FUNCTION_BLOCK AxisVelocityTestSuite 
VAR
	StubAxis : AXIS_REF;
	iStubTask : I_Task;
	TestAxisVelo : MoveVeloTask := (AxisRef := StubAxis);
	ObjTestSuite : TestSuite<TestSuiteParameter.MaxTestCount>('C:\ProgramData\Beckhoff\TwinCAT\3.1\Boot\Object_Tests.xml') := (TestSuiteName := 'Object Test Suite');
END_VAR

DoesTaskAcceptAcceleration_Test();
DoesTaskAcceptDeceleration_Test();
DoesTaskAcceptJerk_Test();
DoesTaskRejectAZeroVelocity_Test();
DoesTaskRejectNegativeAccell_Test();
DoesTaskRejectNegativeDecel_Test();
DoesTaskRejectNegativeJerk_Test();
DoesTaskRejectNegativeVelocity_Test();

METHOD DoesTaskAcceptAcceleration_Test
VAR_INST
	Expected : BOOL := TRUE;
	Actual	 : BOOL;
END_VAR
IF ObjTestSuite.Test(__POUNAME()).ExecuteTest() THEN
	TestAxisVelo.Acceleration := 1.0;
	Actual := TestAxisVelo.Acceleration = 1.0;
	ObjTestSuite.Test(__POUNAME()).AssertEqual(Expected, Actual);
	TestAxisVelo.Acceleration := 0.0;
	TestAxisVelo.Abort();
END_IF
END_METHOD

METHOD DoesTaskAcceptDeceleration_Test
VAR_INST
	Expected : BOOL := TRUE;
	Actual	 : BOOL;
END_VAR
IF ObjTestSuite.Test(__POUNAME()).ExecuteTest() THEN
	TestAxisVelo.Deceleration := 1.0;
	Actual := TestAxisVelo.Deceleration = 1.0;
	ObjTestSuite.Test(__POUNAME()).AssertEqual(Expected, Actual);
	TestAxisVelo.Deceleration := 0.0;
	TestAxisVelo.Abort();
END_IF
END_METHOD

METHOD DoesTaskAcceptJerk_Test
VAR_INST
	Expected : BOOL := TRUE;
	Actual	 : BOOL;
END_VAR
IF ObjTestSuite.Test(__POUNAME()).ExecuteTest() THEN
	TestAxisVelo.Jerk := 1.0;
	Actual := TestAxisVelo.Jerk = 1.0;
	ObjTestSuite.Test(__POUNAME()).AssertEqual(Expected, Actual);
	TestAxisVelo.Jerk := 0.0;
	TestAxisVelo.Abort();
END_IF
END_METHOD

METHOD DoesTaskRejectAZeroVelocity_Test
VAR_INST
	Expected : BOOL := TRUE;
	Actual	 : BOOL;
END_VAR
IF ObjTestSuite.Test(__POUNAME()).ExecuteTest() THEN
	iStubTask := 0;
	Actual := FAILED(TestAxisVelo.MoveAtVelocity(mc_direction.MC_Positive_Direction, 0.0));
	ObjTestSuite.Test(__POUNAME()).AssertEqual(Expected, Actual);
	TestAxisVelo.Abort();
END_IF
END_METHOD

METHOD DoesTaskRejectNegativeAccell_Test
VAR_INST
	Expected : BOOL := TRUE;
	Actual	 : BOOL;
END_VAR
IF ObjTestSuite.Test(__POUNAME()).ExecuteTest() THEN
	TestAxisVelo.Acceleration := -1.0;
	Actual := TestAxisVelo.Acceleration = 0.0;
	ObjTestSuite.Test(__POUNAME()).AssertEqual(Expected, Actual);
	TestAxisVelo.Abort();
END_IF
END_METHOD

METHOD DoesTaskRejectNegativeDecel_Test
VAR_INST
	Expected : BOOL := TRUE;
	Actual	 : BOOL;
END_VAR
IF ObjTestSuite.Test(__POUNAME()).ExecuteTest() THEN
	TestAxisVelo.Deceleration := -1.0;
	Actual := TestAxisVelo.Deceleration = 0.0;
	ObjTestSuite.Test(__POUNAME()).AssertEqual(Expected, Actual);
	TestAxisVelo.Abort();
END_IF
END_METHOD

METHOD DoesTaskRejectNegativeJerk_Test
VAR_INST
	Expected : BOOL := TRUE;
	Actual	 : BOOL;
END_VAR
IF ObjTestSuite.Test(__POUNAME()).ExecuteTest() THEN
	TestAxisVelo.Jerk := -1.0;
	Actual := TestAxisVelo.jerk = 0.0;
	ObjTestSuite.Test(__POUNAME()).AssertEqual(Expected, Actual);
	TestAxisVelo.Abort();
END_IF
END_METHOD

METHOD DoesTaskRejectNegativeVelocity_Test
VAR_INST
	Expected : BOOL := TRUE;
	Actual	 : BOOL;
END_VAR
IF ObjTestSuite.Test(__POUNAME()).ExecuteTest() THEN
	iStubTask := 0;
	Actual := FAILED(TestAxisVelo.MoveAtVelocity(mc_direction.MC_Positive_Direction, -70.0));
	ObjTestSuite.Test(__POUNAME()).AssertEqual(Expected, Actual);
	TestAxisVelo.Abort();
END_IF
END_METHOD

END_FUNCTION_BLOCK

(* stored: Version 1.1.0.1
   POU AxisVelocityTestSuite: Id {6f423009-7ac9-4bbc-9784-ede5e34ea635}, SpecialFunc None
   Method DoesTaskAcceptAcceleration_Test: Id {0d230c75-21d6-4506-bf0c-f778675ad65c}
   Method DoesTaskAcceptDeceleration_Test: Id {a725a69d-9af8-45c5-ad00-c4fbd028eb4f}
   Method DoesTaskAcceptJerk_Test: Id {d560ffe4-245c-4d46-b643-11f6f65f8005}
   Method DoesTaskRejectAZeroVelocity_Test: Id {9233b2c1-1cb2-4bb5-b278-086baa3c1d61}
   Method DoesTaskRejectNegativeAccell_Test: Id {d4be8287-9832-4973-8435-cd5c515b6477}
   Method DoesTaskRejectNegativeDecel_Test: Id {0423d667-7b84-4a25-8f3d-e1a2d4aba3b5}
   Method DoesTaskRejectNegativeJerk_Test: Id {ddb0c839-acfd-4f35-93b9-46f24cb5f745}
   Method DoesTaskRejectNegativeVelocity_Test: Id {12aaa02a-5789-47ac-aae9-1dcdc1d6405e} *)
